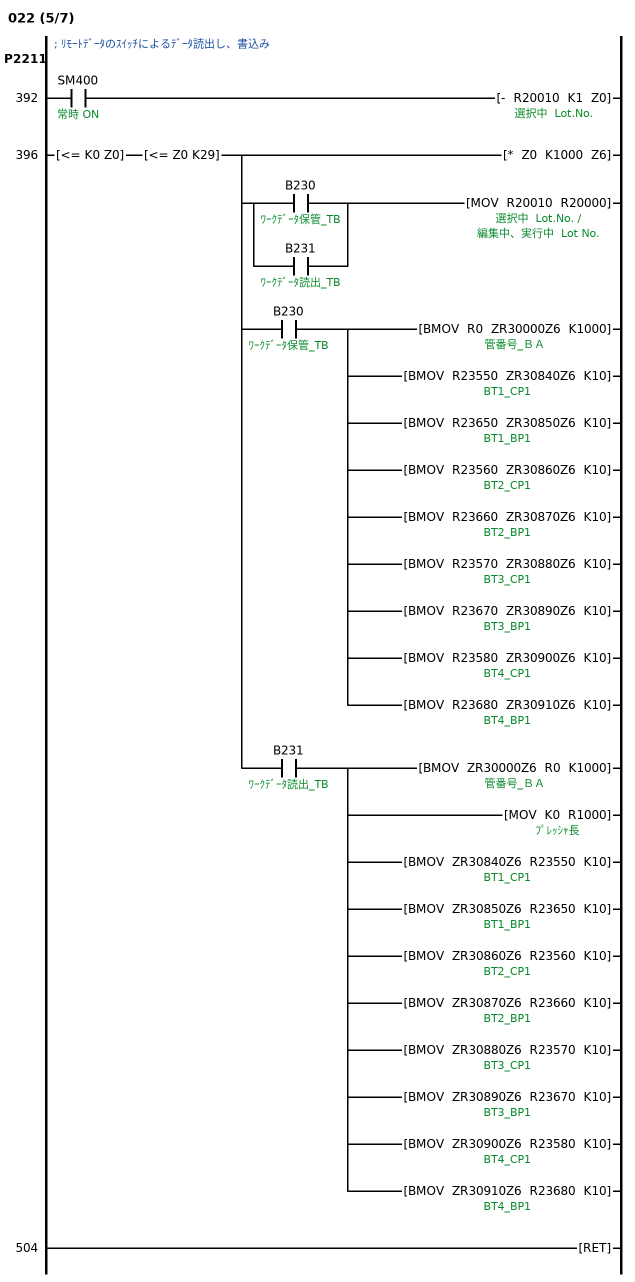
392   LD      SM400  ; 常時 ON
      -       R20010 K1 Z0
396   LD<=    K0 Z0
      AND<=   Z0 K29
      *       Z0 K1000 Z6
      MPS
      LD      B230  ; ﾜｰｸﾃﾞｰﾀ保管_TB
      OR      B231  ; ﾜｰｸﾃﾞｰﾀ読出_TB
      ANB
      MOV     R20010 R20000
      MRD
      AND     B230  ; ﾜｰｸﾃﾞｰﾀ保管_TB
      BMOV    R0 ZR30000Z6 K1000
      BMOV    R23550 ZR30840Z6 K10
      BMOV    R23650 ZR30850Z6 K10
      BMOV    R23560 ZR30860Z6 K10
      BMOV    R23660 ZR30870Z6 K10
      BMOV    R23570 ZR30880Z6 K10
      BMOV    R23670 ZR30890Z6 K10
      BMOV    R23580 ZR30900Z6 K10
      BMOV    R23680 ZR30910Z6 K10
      MPP
      AND     B231  ; ﾜｰｸﾃﾞｰﾀ読出_TB
      BMOV    ZR30000Z6 R0 K1000
      MOV     K0 R1000
      BMOV    ZR30840Z6 R23550 K10
      BMOV    ZR30850Z6 R23650 K10
      BMOV    ZR30860Z6 R23560 K10
      BMOV    ZR30870Z6 R23660 K10
      BMOV    ZR30880Z6 R23570 K10
      BMOV    ZR30890Z6 R23670 K10
      BMOV    ZR30900Z6 R23580 K10
      BMOV    ZR30910Z6 R23680 K10
504   RET
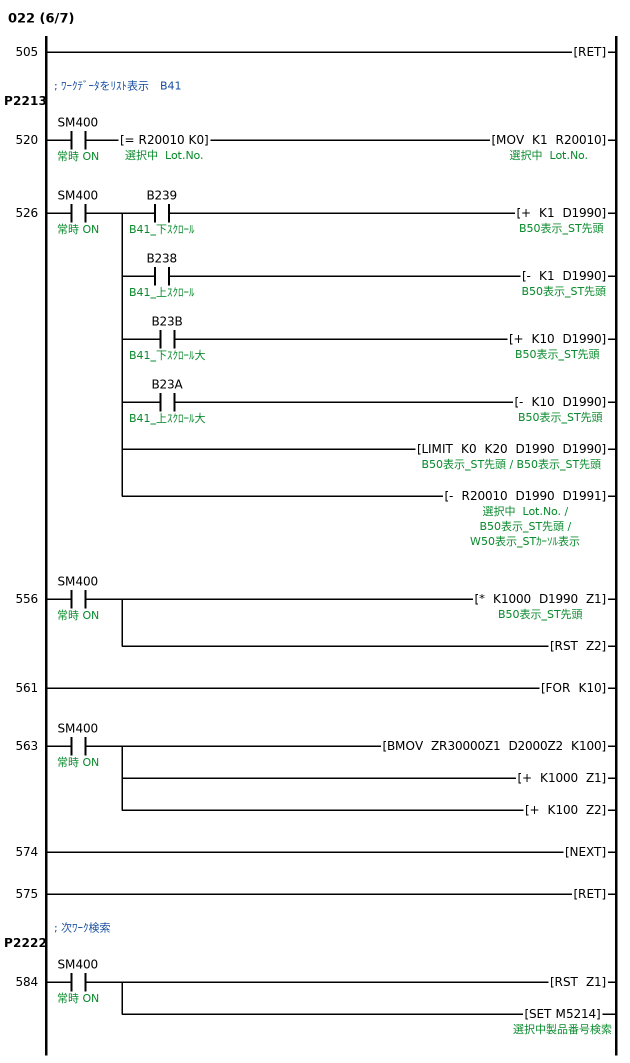
505   RET
; ﾜｰｸﾃﾞｰﾀをﾘｽﾄ表示　B41
      P2213
520   LD      SM400  ; 常時 ON
      AND=    R20010 K0  ; 選択中  Lot.No.
      MOV     K1 R20010
526   LD      SM400  ; 常時 ON
      MPS
      AND     B239  ; B41_下ｽｸﾛｰﾙ
      +       K1 D1990
      MRD
      AND     B238  ; B41_上ｽｸﾛｰﾙ
      -       K1 D1990
      MRD
      AND     B23B  ; B41_下ｽｸﾛｰﾙ大
      +       K10 D1990
      MRD
      AND     B23A  ; B41_上ｽｸﾛｰﾙ大
      -       K10 D1990
      MPP
      LIMIT   K0 K20 D1990 D1990
      -       R20010 D1990 D1991
556   LD      SM400  ; 常時 ON
      *       K1000 D1990 Z1
      RST     Z2
561   FOR     K10
563   LD      SM400  ; 常時 ON
      BMOV    ZR30000Z1 D2000Z2 K100
      +       K1000 Z1
      +       K100 Z2
574   NEXT
575   RET
; 次ﾜｰｸ検索
      P2222
584   LD      SM400  ; 常時 ON
      RST     Z1
      SET     M5214  ; 選択中製品番号検索
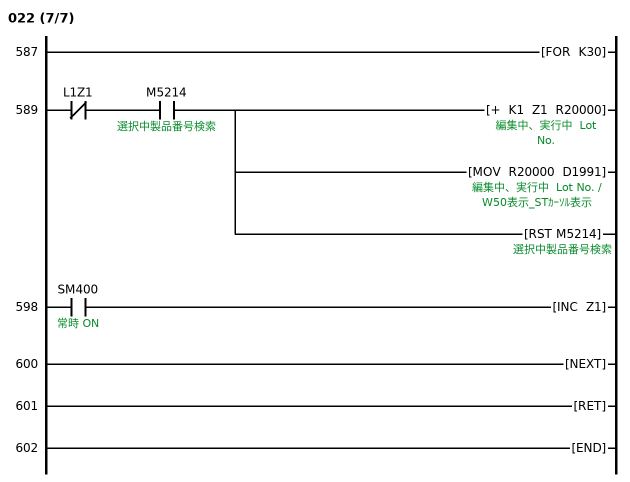
587   FOR     K30
589   LDI     L1Z1
      AND     M5214  ; 選択中製品番号検索
      +       K1 Z1 R20000
      MOV     R20000 D1991
      RST     M5214  ; 選択中製品番号検索
598   LD      SM400  ; 常時 ON
      INC     Z1
600   NEXT
601   RET
602   END
END_PROGRAM

PROGRAM 023  // ﾃﾞｰﾀﾁｪｯｸ
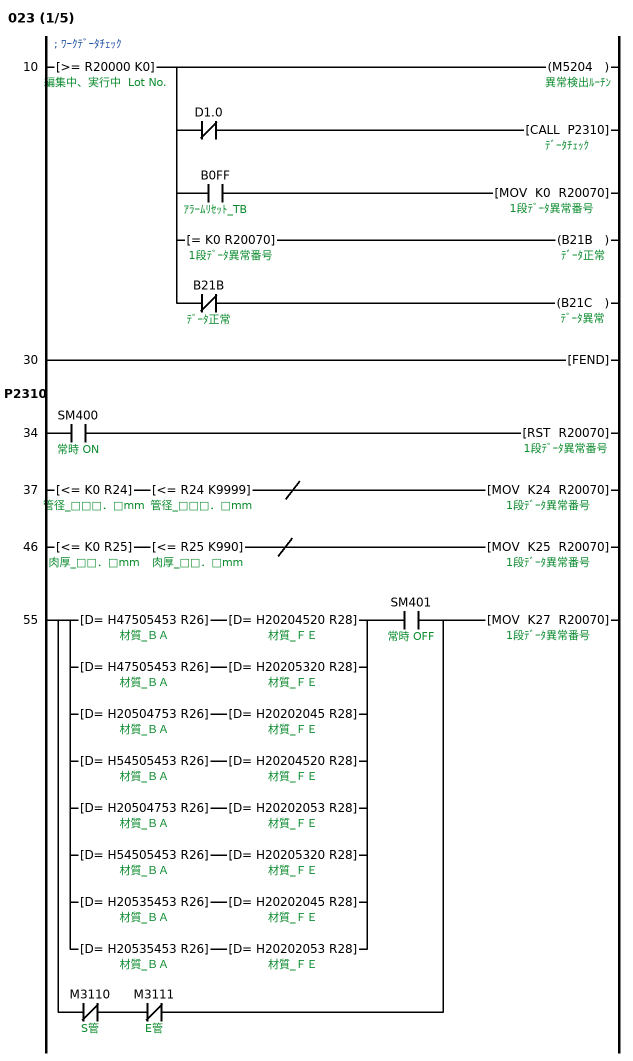
; 
; ﾜｰｸﾃﾞｰﾀﾁｪｯｸ
10    LD>=    R20000 K0  ; 編集中、実行中  Lot No.
      OUT     M5204  ; 異常検出ﾙｰﾁﾝ
      MPS
      ANI     D1.0
      CALL    P2310  ; ﾃﾞｰﾀﾁｪｯｸ
      MRD
      AND     B0FF  ; ｱﾗｰﾑﾘｾｯﾄ_TB
      MOV     K0 R20070  ; 1段ﾃﾞｰﾀ異常番号
      MRD
      AND=    K0 R20070  ; 1段ﾃﾞｰﾀ異常番号
      OUT     B21B  ; ﾃﾞｰﾀ正常
      MPP
      ANI     B21B  ; ﾃﾞｰﾀ正常
      OUT     B21C  ; ﾃﾞｰﾀ異常
30    FEND
; 
      P2310
34    LD      SM400  ; 常時 ON
      RST     R20070  ; 1段ﾃﾞｰﾀ異常番号
37    LD<=    K0 R24  ; 管径_□□□．□mm
      AND<=   R24 K9999  ; 管径_□□□．□mm
      INV
      MOV     K24 R20070
46    LD<=    K0 R25  ; 肉厚_□□．□mm
      AND<=   R25 K990  ; 肉厚_□□．□mm
      INV
      MOV     K25 R20070
55    LDD=    H47505453 R26  ; 材質_ＢＡ
      ANDD=   H20204520 R28  ; 材質_ＦＥ
      LDD=    H47505453 R26  ; 材質_ＢＡ
      ANDD=   H20205320 R28  ; 材質_ＦＥ
      ORB
      LDD=    H20504753 R26  ; 材質_ＢＡ
      ANDD=   H20202045 R28  ; 材質_ＦＥ
      ORB
      LDD=    H54505453 R26  ; 材質_ＢＡ
      ANDD=   H20204520 R28  ; 材質_ＦＥ
      ORB
      LDD=    H20504753 R26  ; 材質_ＢＡ
      ANDD=   H20202053 R28  ; 材質_ＦＥ
      ORB
      LDD=    H54505453 R26  ; 材質_ＢＡ
      ANDD=   H20205320 R28  ; 材質_ＦＥ
      ORB
      LDD=    H20535453 R26  ; 材質_ＢＡ
      ANDD=   H20202045 R28  ; 材質_ＦＥ
      ORB
      LDD=    H20535453 R26  ; 材質_ＢＡ
      ANDD=   H20202053 R28  ; 材質_ＦＥ
      ORB
      AND     SM401  ; 常時 OFF
      LDI     M3110  ; S管
      ANI     M3111  ; E管
      ORB
      MOV     K27 R20070
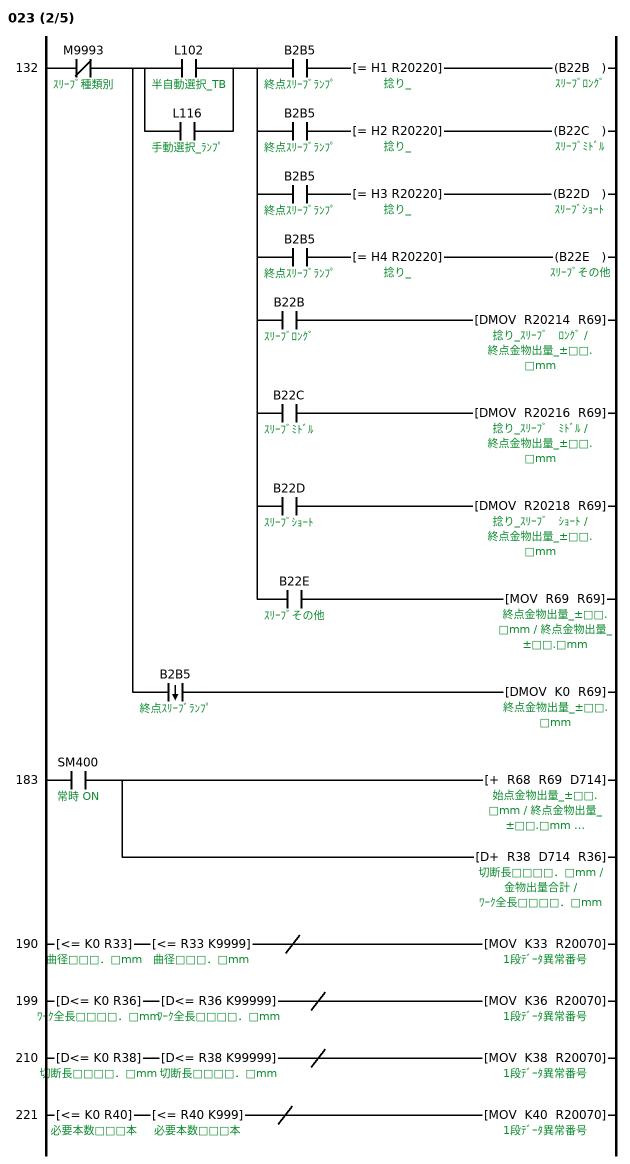
132   LDI     M9993  ; ｽﾘｰﾌﾞ種類別
      MPS
      LD      L102  ; 半自動選択_TB
      OR      L116  ; 手動選択_ﾗﾝﾌﾟ
      ANB
      MPS
      AND     B2B5  ; 終点ｽﾘｰﾌﾞﾗﾝﾌﾟ
      AND=    H1 R20220  ; 捻り_
      OUT     B22B  ; ｽﾘｰﾌﾞﾛﾝｸﾞ
      MRD
      AND     B2B5  ; 終点ｽﾘｰﾌﾞﾗﾝﾌﾟ
      AND=    H2 R20220  ; 捻り_
      OUT     B22C  ; ｽﾘｰﾌﾞﾐﾄﾞﾙ
      MRD
      AND     B2B5  ; 終点ｽﾘｰﾌﾞﾗﾝﾌﾟ
      AND=    H3 R20220  ; 捻り_
      OUT     B22D  ; ｽﾘｰﾌﾞｼｮｰﾄ
      MRD
      AND     B2B5  ; 終点ｽﾘｰﾌﾞﾗﾝﾌﾟ
      AND=    H4 R20220  ; 捻り_
      OUT     B22E  ; ｽﾘｰﾌﾞその他
      MRD
      AND     B22B  ; ｽﾘｰﾌﾞﾛﾝｸﾞ
      DMOV    R20214 R69  ; 捻り_ｽﾘｰﾌﾞ　ﾛﾝｸﾞ / 終点金物出量_±□□.□mm
      MRD
      AND     B22C  ; ｽﾘｰﾌﾞﾐﾄﾞﾙ
      DMOV    R20216 R69  ; 捻り_ｽﾘｰﾌﾞ　ﾐﾄﾞﾙ
      MRD
      AND     B22D  ; ｽﾘｰﾌﾞｼｮｰﾄ
      DMOV    R20218 R69  ; 捻り_ｽﾘｰﾌﾞ　ｼｮｰﾄ
      MPP
      AND     B22E  ; ｽﾘｰﾌﾞその他
      MOV     R69 R69
      MPP
      ANDF    B2B5  ; 終点ｽﾘｰﾌﾞﾗﾝﾌﾟ
      DMOV    K0 R69
183   LD      SM400  ; 常時 ON
      +       R68 R69 D714  ; 始点金物出量_±□□.□mm / 金物出量合計
      D+      R38 D714 R36  ; 切断長□□□□．□mm / ﾜｰｸ全長□□□□．□mm
190   LD<=    K0 R33  ; 曲径□□□．□mm
      AND<=   R33 K9999  ; 曲径□□□．□mm
      INV
      MOV     K33 R20070
199   LDD<=   K0 R36  ; ﾜｰｸ全長□□□□．□mm
      ANDD<=  R36 K99999  ; ﾜｰｸ全長□□□□．□mm
      INV
      MOV     K36 R20070
210   LDD<=   K0 R38  ; 切断長□□□□．□mm
      ANDD<=  R38 K99999  ; 切断長□□□□．□mm
      INV
      MOV     K38 R20070
221   LD<=    K0 R40  ; 必要本数□□□本
      AND<=   R40 K999  ; 必要本数□□□本
      INV
      MOV     K40 R20070
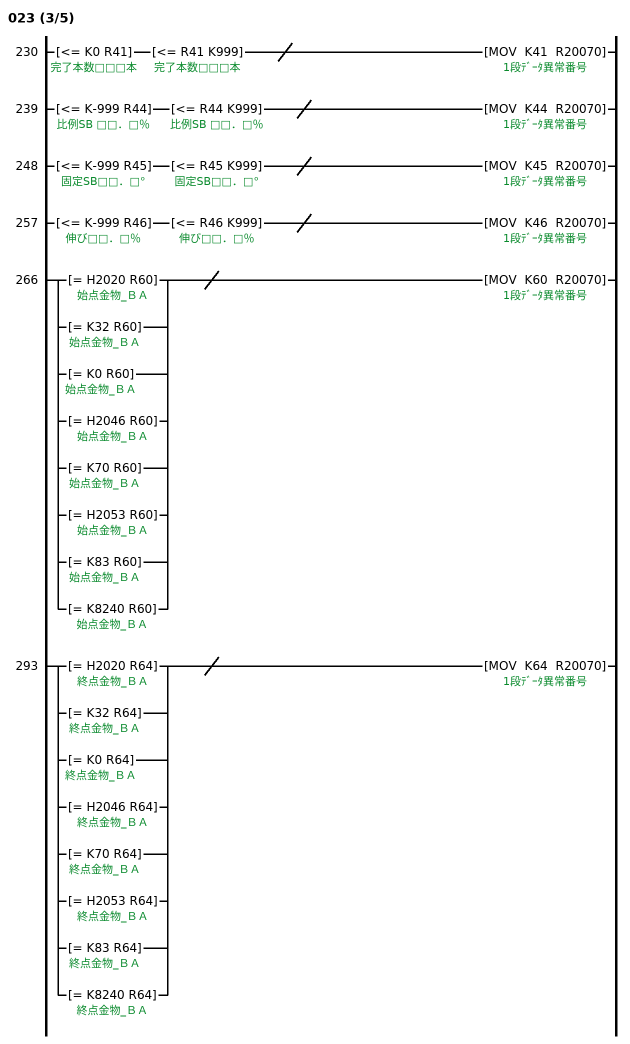
230   LD<=    K0 R41  ; 完了本数□□□本
      AND<=   R41 K999  ; 完了本数□□□本
      INV
      MOV     K41 R20070
239   LD<=    K-999 R44  ; 比例SB □□．□％
      AND<=   R44 K999  ; 比例SB □□．□％
      INV
      MOV     K44 R20070
248   LD<=    K-999 R45  ; 固定SB□□．□°
      AND<=   R45 K999  ; 固定SB□□．□°
      INV
      MOV     K45 R20070
257   LD<=    K-999 R46  ; 伸び□□．□％
      AND<=   R46 K999  ; 伸び□□．□％
      INV
      MOV     K46 R20070
266   LD=     H2020 R60  ; 始点金物_ＢＡ
      OR=     K32 R60  ; 始点金物_ＢＡ
      OR=     K0 R60  ; 始点金物_ＢＡ
      OR=     H2046 R60  ; 始点金物_ＢＡ
      OR=     K70 R60  ; 始点金物_ＢＡ
      OR=     H2053 R60  ; 始点金物_ＢＡ
      OR=     K83 R60  ; 始点金物_ＢＡ
      OR=     K8240 R60  ; 始点金物_ＢＡ
      INV
      MOV     K60 R20070
293   LD=     H2020 R64  ; 終点金物_ＢＡ
      OR=     K32 R64  ; 終点金物_ＢＡ
      OR=     K0 R64  ; 終点金物_ＢＡ
      OR=     H2046 R64  ; 終点金物_ＢＡ
      OR=     K70 R64  ; 終点金物_ＢＡ
      OR=     H2053 R64  ; 終点金物_ＢＡ
      OR=     K83 R64  ; 終点金物_ＢＡ
      OR=     K8240 R64  ; 終点金物_ＢＡ
      INV
      MOV     K64 R20070
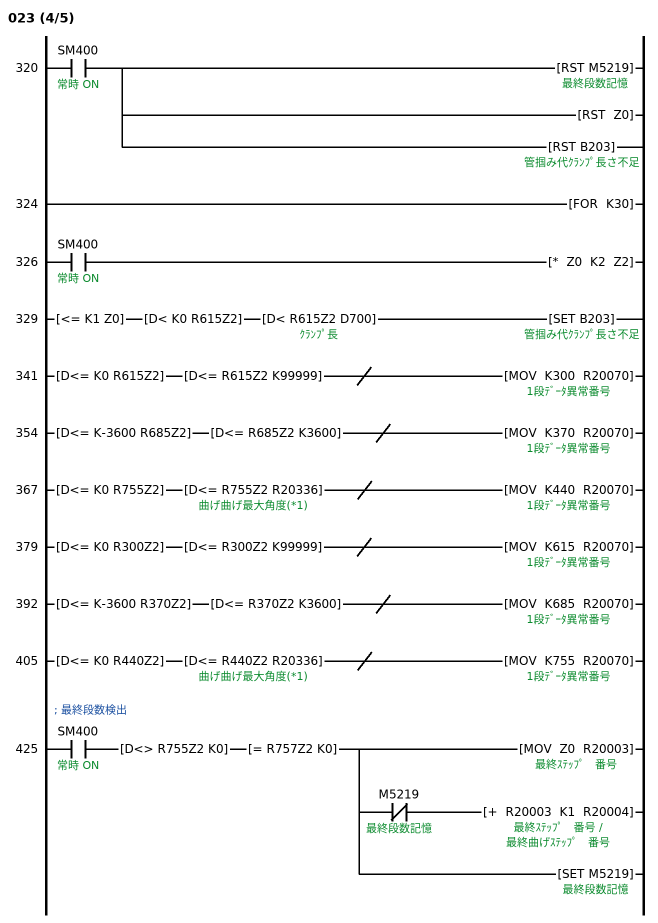
320   LD      SM400  ; 常時 ON
      RST     M5219  ; 最終段数記憶
      RST     Z0
      RST     B203  ; 管掴み代ｸﾗﾝﾌﾟ長さ不足
324   FOR     K30
326   LD      SM400  ; 常時 ON
      *       Z0 K2 Z2
329   LD<=    K1 Z0
      ANDD<   K0 R615Z2
      ANDD<   R615Z2 D700  ; ｸﾗﾝﾌﾟ長
      SET     B203  ; 管掴み代ｸﾗﾝﾌﾟ長さ不足
341   LDD<=   K0 R615Z2
      ANDD<=  R615Z2 K99999
      INV
      MOV     K300 R20070
354   LDD<=   K-3600 R685Z2
      ANDD<=  R685Z2 K3600
      INV
      MOV     K370 R20070
367   LDD<=   K0 R755Z2
      ANDD<=  R755Z2 R20336  ; 曲げ曲げ最大角度(*1)
      INV
      MOV     K440 R20070
379   LDD<=   K0 R300Z2
      ANDD<=  R300Z2 K99999
      INV
      MOV     K615 R20070
392   LDD<=   K-3600 R370Z2
      ANDD<=  R370Z2 K3600
      INV
      MOV     K685 R20070
405   LDD<=   K0 R440Z2
      ANDD<=  R440Z2 R20336  ; 曲げ曲げ最大角度(*1)
      INV
      MOV     K755 R20070
; 最終段数検出
425   LD      SM400  ; 常時 ON
      ANDD<>  R755Z2 K0
      AND=    R757Z2 K0
      MOV     Z0 R20003  ; 最終ｽﾃｯﾌﾟ   番号
      MPS
      ANI     M5219  ; 最終段数記憶
      +       R20003 K1 R20004  ; 最終曲げｽﾃｯﾌﾟ   番号
      MPP
      SET     M5219  ; 最終段数記憶
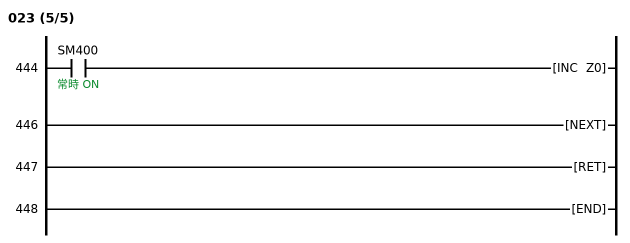
444   LD      SM400  ; 常時 ON
      INC     Z0
446   NEXT
447   RET
448   END
END_PROGRAM

PROGRAM 025  // 完了表示とPC通信
; 完了表示＊Ｙ付加
      P2500
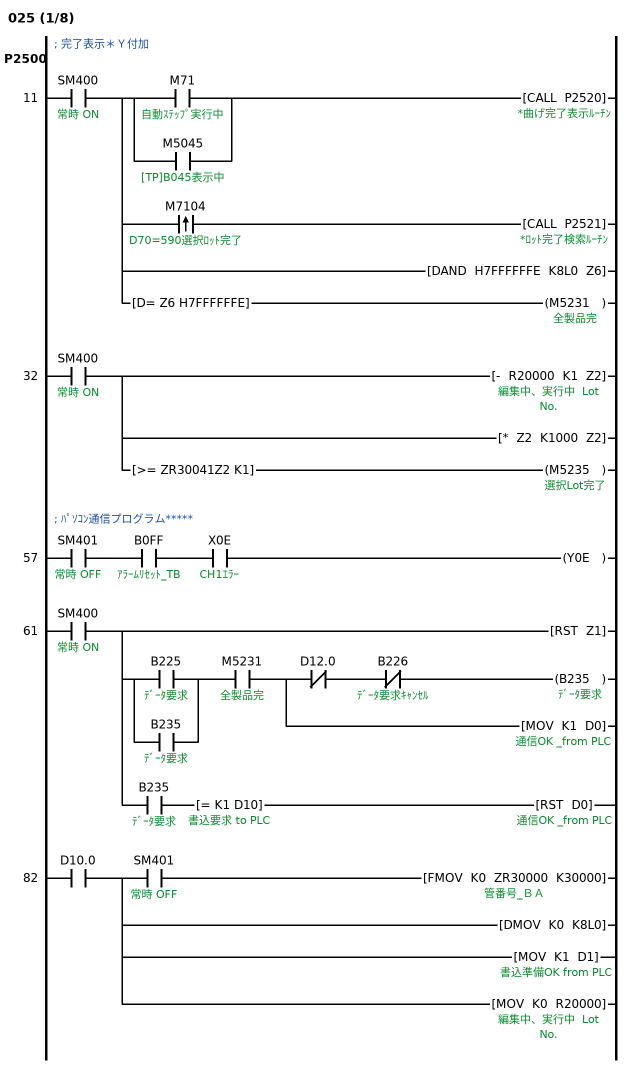
11    LD      SM400  ; 常時 ON
      MPS
      LD      M71  ; 自動ｽﾃｯﾌﾟ実行中
      OR      M5045  ; [TP]B045表示中
      ANB
      CALL    P2520  ; *曲げ完了表示ﾙｰﾁﾝ
      MRD
      ANDP    M7104  ; D70=590選択ﾛｯﾄ完了
      CALL    P2521  ; *ﾛｯﾄ完了検索ﾙｰﾁﾝ
      MPP
      DAND    H7FFFFFFE K8L0 Z6
      ANDD=   Z6 H7FFFFFFE
      OUT     M5231  ; 全製品完
32    LD      SM400  ; 常時 ON
      -       R20000 K1 Z2  ; 編集中、実行中  Lot No.
      *       Z2 K1000 Z2
      AND>=   ZR30041Z2 K1
      OUT     M5235  ; 選択Lot完了
; ﾊﾟｿｺﾝ通信プログラム*****
57    LD      SM401  ; 常時 OFF
      AND     B0FF  ; ｱﾗｰﾑﾘｾｯﾄ_TB
      AND     X0E  ; CH1ｴﾗｰ
      OUT     Y0E
61    LD      SM400  ; 常時 ON
      RST     Z1
      MPS
      LD      B225  ; ﾃﾞｰﾀ要求
      OR      B235  ; ﾃﾞｰﾀ要求
      ANB
      AND     M5231  ; 全製品完
      MPS
      ANI     D12.0
      ANI     B226  ; ﾃﾞｰﾀ要求ｷｬﾝｾﾙ
      OUT     B235  ; ﾃﾞｰﾀ要求
      MPP
      MOV     K1 D0  ; 通信OK _from PLC
      MPP
      AND     B235  ; ﾃﾞｰﾀ要求
      AND=    K1 D10  ; 書込要求 to PLC
      RST     D0  ; 通信OK _from PLC
82    LD      D10.0
      MPS
      AND     SM401  ; 常時 OFF
      FMOV    K0 ZR30000 K30000  ; 管番号_ＢＡ
      MPP
      DMOV    K0 K8L0
      MOV     K1 D1  ; 書込準備OK from PLC
      MOV     K0 R20000
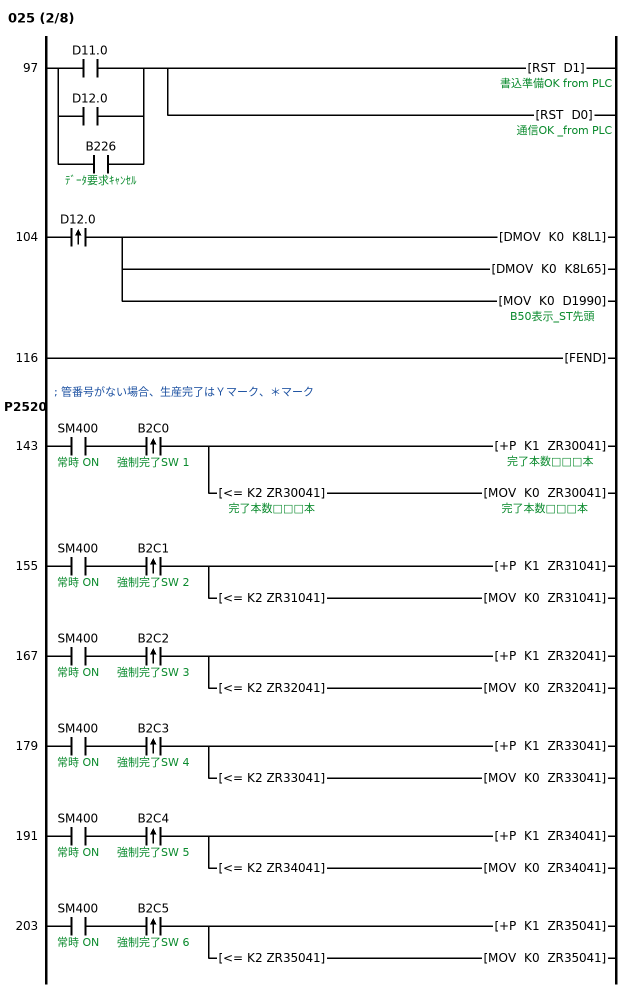
97    LD      D11.0
      OR      D12.0
      OR      B226  ; ﾃﾞｰﾀ要求ｷｬﾝｾﾙ
      RST     D1  ; 書込準備OK from PLC
      RST     D0  ; 通信OK _from PLC
104   LDP     D12.0
      DMOV    K0 K8L1  ; ﾛｯﾄ№-01作業完了
      DMOV    K0 K8L65  ; ﾛｯﾄ№-01作業完了記憶
      MOV     K0 D1990  ; B50表示_ST先頭
116   FEND
; 管番号がない場合、生産完了はＹマーク、＊マーク
      P2520
143   LD      SM400  ; 常時 ON
      ANDP    B2C0  ; 強制完了SW 1
      +P      K1 ZR30041  ; 完了本数□□□本
      AND<=   K2 ZR30041  ; 完了本数□□□本
      MOV     K0 ZR30041
155   LD      SM400  ; 常時 ON
      ANDP    B2C1  ; 強制完了SW 2
      +P      K1 ZR31041
      AND<=   K2 ZR31041
      MOV     K0 ZR31041
167   LD      SM400  ; 常時 ON
      ANDP    B2C2  ; 強制完了SW 3
      +P      K1 ZR32041
      AND<=   K2 ZR32041
      MOV     K0 ZR32041
179   LD      SM400  ; 常時 ON
      ANDP    B2C3  ; 強制完了SW 4
      +P      K1 ZR33041
      AND<=   K2 ZR33041
      MOV     K0 ZR33041
191   LD      SM400  ; 常時 ON
      ANDP    B2C4  ; 強制完了SW 5
      +P      K1 ZR34041
      AND<=   K2 ZR34041
      MOV     K0 ZR34041
203   LD      SM400  ; 常時 ON
      ANDP    B2C5  ; 強制完了SW 6
      +P      K1 ZR35041
      AND<=   K2 ZR35041
      MOV     K0 ZR35041
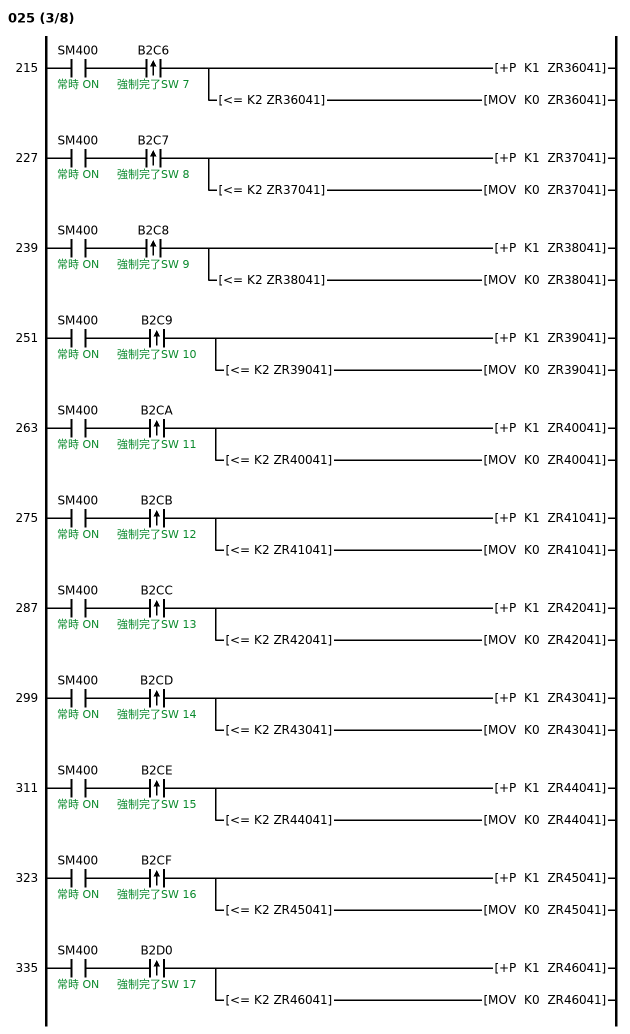
215   LD      SM400  ; 常時 ON
      ANDP    B2C6  ; 強制完了SW 7
      +P      K1 ZR36041
      AND<=   K2 ZR36041
      MOV     K0 ZR36041
227   LD      SM400  ; 常時 ON
      ANDP    B2C7  ; 強制完了SW 8
      +P      K1 ZR37041
      AND<=   K2 ZR37041
      MOV     K0 ZR37041
239   LD      SM400  ; 常時 ON
      ANDP    B2C8  ; 強制完了SW 9
      +P      K1 ZR38041
      AND<=   K2 ZR38041
      MOV     K0 ZR38041
251   LD      SM400  ; 常時 ON
      ANDP    B2C9  ; 強制完了SW 10
      +P      K1 ZR39041
      AND<=   K2 ZR39041
      MOV     K0 ZR39041
263   LD      SM400  ; 常時 ON
      ANDP    B2CA  ; 強制完了SW 11
      +P      K1 ZR40041
      AND<=   K2 ZR40041
      MOV     K0 ZR40041
275   LD      SM400  ; 常時 ON
      ANDP    B2CB  ; 強制完了SW 12
      +P      K1 ZR41041
      AND<=   K2 ZR41041
      MOV     K0 ZR41041
287   LD      SM400  ; 常時 ON
      ANDP    B2CC  ; 強制完了SW 13
      +P      K1 ZR42041
      AND<=   K2 ZR42041
      MOV     K0 ZR42041
299   LD      SM400  ; 常時 ON
      ANDP    B2CD  ; 強制完了SW 14
      +P      K1 ZR43041
      AND<=   K2 ZR43041
      MOV     K0 ZR43041
311   LD      SM400  ; 常時 ON
      ANDP    B2CE  ; 強制完了SW 15
      +P      K1 ZR44041
      AND<=   K2 ZR44041
      MOV     K0 ZR44041
323   LD      SM400  ; 常時 ON
      ANDP    B2CF  ; 強制完了SW 16
      +P      K1 ZR45041
      AND<=   K2 ZR45041
      MOV     K0 ZR45041
335   LD      SM400  ; 常時 ON
      ANDP    B2D0  ; 強制完了SW 17
      +P      K1 ZR46041
      AND<=   K2 ZR46041
      MOV     K0 ZR46041
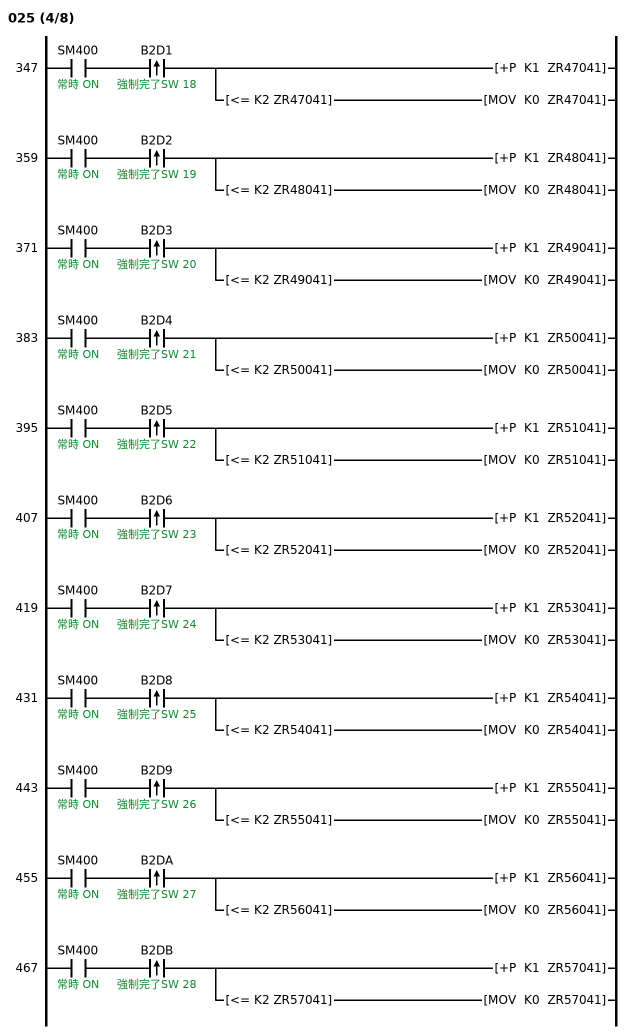
347   LD      SM400  ; 常時 ON
      ANDP    B2D1  ; 強制完了SW 18
      +P      K1 ZR47041
      AND<=   K2 ZR47041
      MOV     K0 ZR47041
359   LD      SM400  ; 常時 ON
      ANDP    B2D2  ; 強制完了SW 19
      +P      K1 ZR48041
      AND<=   K2 ZR48041
      MOV     K0 ZR48041
371   LD      SM400  ; 常時 ON
      ANDP    B2D3  ; 強制完了SW 20
      +P      K1 ZR49041
      AND<=   K2 ZR49041
      MOV     K0 ZR49041
383   LD      SM400  ; 常時 ON
      ANDP    B2D4  ; 強制完了SW 21
      +P      K1 ZR50041
      AND<=   K2 ZR50041
      MOV     K0 ZR50041
395   LD      SM400  ; 常時 ON
      ANDP    B2D5  ; 強制完了SW 22
      +P      K1 ZR51041
      AND<=   K2 ZR51041
      MOV     K0 ZR51041
407   LD      SM400  ; 常時 ON
      ANDP    B2D6  ; 強制完了SW 23
      +P      K1 ZR52041
      AND<=   K2 ZR52041
      MOV     K0 ZR52041
419   LD      SM400  ; 常時 ON
      ANDP    B2D7  ; 強制完了SW 24
      +P      K1 ZR53041
      AND<=   K2 ZR53041
      MOV     K0 ZR53041
431   LD      SM400  ; 常時 ON
      ANDP    B2D8  ; 強制完了SW 25
      +P      K1 ZR54041
      AND<=   K2 ZR54041
      MOV     K0 ZR54041
443   LD      SM400  ; 常時 ON
      ANDP    B2D9  ; 強制完了SW 26
      +P      K1 ZR55041
      AND<=   K2 ZR55041
      MOV     K0 ZR55041
455   LD      SM400  ; 常時 ON
      ANDP    B2DA  ; 強制完了SW 27
      +P      K1 ZR56041
      AND<=   K2 ZR56041
      MOV     K0 ZR56041
467   LD      SM400  ; 常時 ON
      ANDP    B2DB  ; 強制完了SW 28
      +P      K1 ZR57041
      AND<=   K2 ZR57041
      MOV     K0 ZR57041
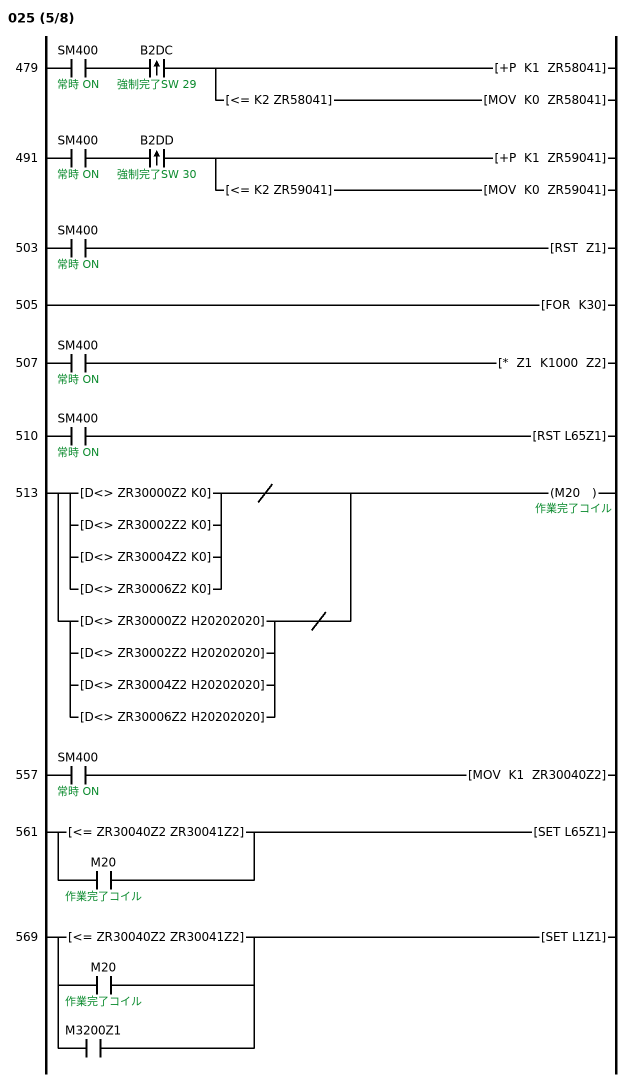
479   LD      SM400  ; 常時 ON
      ANDP    B2DC  ; 強制完了SW 29
      +P      K1 ZR58041
      AND<=   K2 ZR58041
      MOV     K0 ZR58041
491   LD      SM400  ; 常時 ON
      ANDP    B2DD  ; 強制完了SW 30
      +P      K1 ZR59041
      AND<=   K2 ZR59041
      MOV     K0 ZR59041
503   LD      SM400  ; 常時 ON
      RST     Z1
505   FOR     K30
507   LD      SM400  ; 常時 ON
      *       Z1 K1000 Z2
510   LD      SM400  ; 常時 ON
      RST     L65Z1
513   LDD<>   ZR30000Z2 K0
      ORD<>   ZR30002Z2 K0
      ORD<>   ZR30004Z2 K0
      ORD<>   ZR30006Z2 K0
      INV
      LDD<>   ZR30000Z2 H20202020
      ORD<>   ZR30002Z2 H20202020
      ORD<>   ZR30004Z2 H20202020
      ORD<>   ZR30006Z2 H20202020
      INV
      ORB
      OUT     M20  ; 作業完了コイル
557   LD      SM400  ; 常時 ON
      MOV     K1 ZR30040Z2
561   LD<=    ZR30040Z2 ZR30041Z2
      OR      M20  ; 作業完了コイル
      SET     L65Z1
569   LD<=    ZR30040Z2 ZR30041Z2
      OR      M20  ; 作業完了コイル
      OR      M3200Z1
      SET     L1Z1
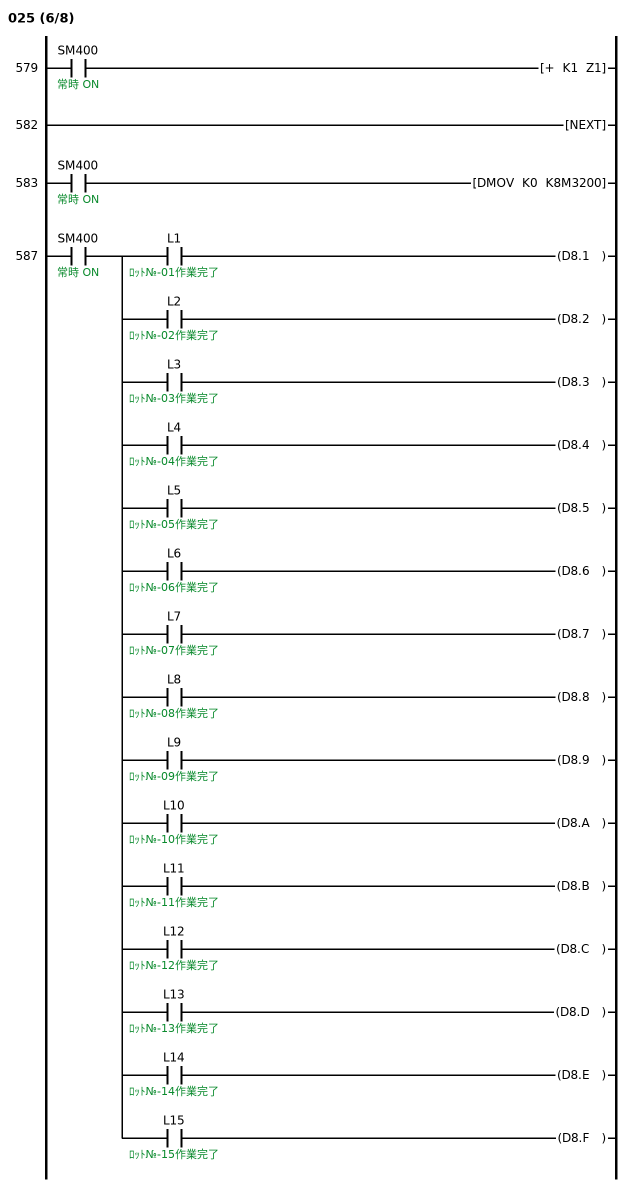
579   LD      SM400  ; 常時 ON
      +       K1 Z1
582   NEXT
583   LD      SM400  ; 常時 ON
      DMOV    K0 K8M3200  ; ﾛｯﾄNo.-01作業完了
587   LD      SM400  ; 常時 ON
      MPS
      AND     L1  ; ﾛｯﾄ№-01作業完了
      OUT     D8.1
      MRD
      AND     L2  ; ﾛｯﾄ№-02作業完了
      OUT     D8.2
      MRD
      AND     L3  ; ﾛｯﾄ№-03作業完了
      OUT     D8.3
      MRD
      AND     L4  ; ﾛｯﾄ№-04作業完了
      OUT     D8.4
      MRD
      AND     L5  ; ﾛｯﾄ№-05作業完了
      OUT     D8.5
      MRD
      AND     L6  ; ﾛｯﾄ№-06作業完了
      OUT     D8.6
      MRD
      AND     L7  ; ﾛｯﾄ№-07作業完了
      OUT     D8.7
      MRD
      AND     L8  ; ﾛｯﾄ№-08作業完了
      OUT     D8.8
      MRD
      AND     L9  ; ﾛｯﾄ№-09作業完了
      OUT     D8.9
      MRD
      AND     L10  ; ﾛｯﾄ№-10作業完了
      OUT     D8.A
      MRD
      AND     L11  ; ﾛｯﾄ№-11作業完了
      OUT     D8.B
      MRD
      AND     L12  ; ﾛｯﾄ№-12作業完了
      OUT     D8.C
      MRD
      AND     L13  ; ﾛｯﾄ№-13作業完了
      OUT     D8.D
      MRD
      AND     L14  ; ﾛｯﾄ№-14作業完了
      OUT     D8.E
      MPP
      AND     L15  ; ﾛｯﾄ№-15作業完了
      OUT     D8.F
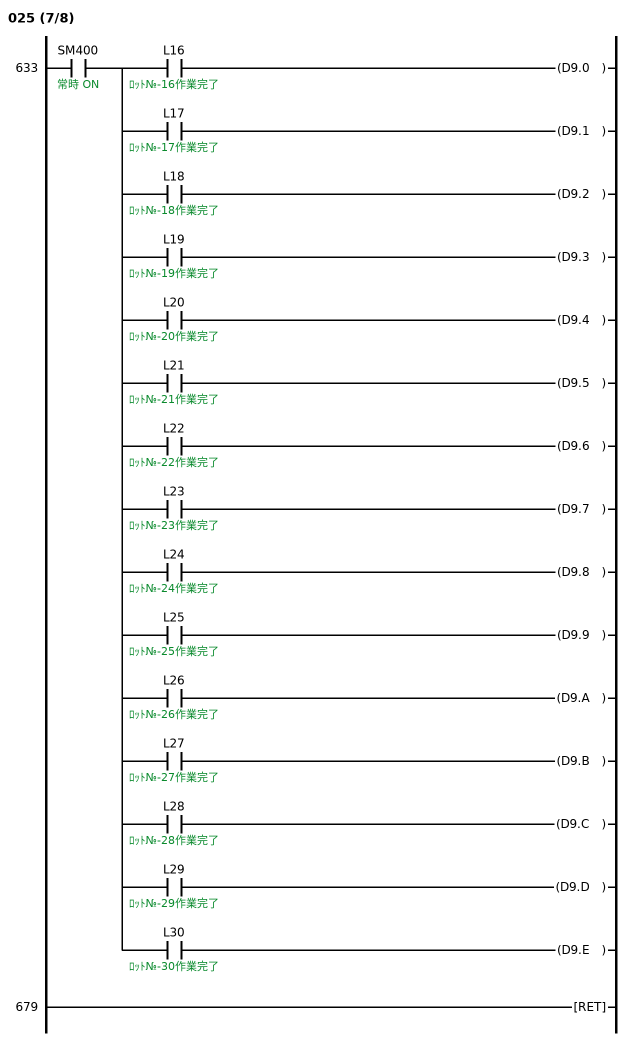
633   LD      SM400  ; 常時 ON
      MPS
      AND     L16  ; ﾛｯﾄ№-16作業完了
      OUT     D9.0
      MRD
      AND     L17  ; ﾛｯﾄ№-17作業完了
      OUT     D9.1
      MRD
      AND     L18  ; ﾛｯﾄ№-18作業完了
      OUT     D9.2
      MRD
      AND     L19  ; ﾛｯﾄ№-19作業完了
      OUT     D9.3
      MRD
      AND     L20  ; ﾛｯﾄ№-20作業完了
      OUT     D9.4
      MRD
      AND     L21  ; ﾛｯﾄ№-21作業完了
      OUT     D9.5
      MRD
      AND     L22  ; ﾛｯﾄ№-22作業完了
      OUT     D9.6
      MRD
      AND     L23  ; ﾛｯﾄ№-23作業完了
      OUT     D9.7
      MRD
      AND     L24  ; ﾛｯﾄ№-24作業完了
      OUT     D9.8
      MRD
      AND     L25  ; ﾛｯﾄ№-25作業完了
      OUT     D9.9
      MRD
      AND     L26  ; ﾛｯﾄ№-26作業完了
      OUT     D9.A
      MRD
      AND     L27  ; ﾛｯﾄ№-27作業完了
      OUT     D9.B
      MRD
      AND     L28  ; ﾛｯﾄ№-28作業完了
      OUT     D9.C
      MRD
      AND     L29  ; ﾛｯﾄ№-29作業完了
      OUT     D9.D
      MPP
      AND     L30  ; ﾛｯﾄ№-30作業完了
      OUT     D9.E
679   RET
; 生産本数分完了で完了マーク
      P2521
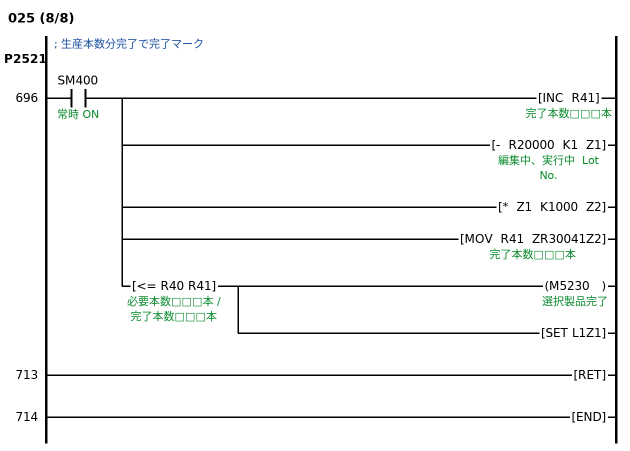
696   LD      SM400  ; 常時 ON
      INC     R41  ; 完了本数□□□本
      -       R20000 K1 Z1
      *       Z1 K1000 Z2
      MOV     R41 ZR30041Z2
      AND<=   R40 R41  ; 必要本数□□□本 / 完了本数□□□本
      OUT     M5230  ; 選択製品完了
      SET     L1Z1
713   RET
714   END
END_PROGRAM

PROGRAM 027  // 管径別ﾃﾞｰﾀ検索
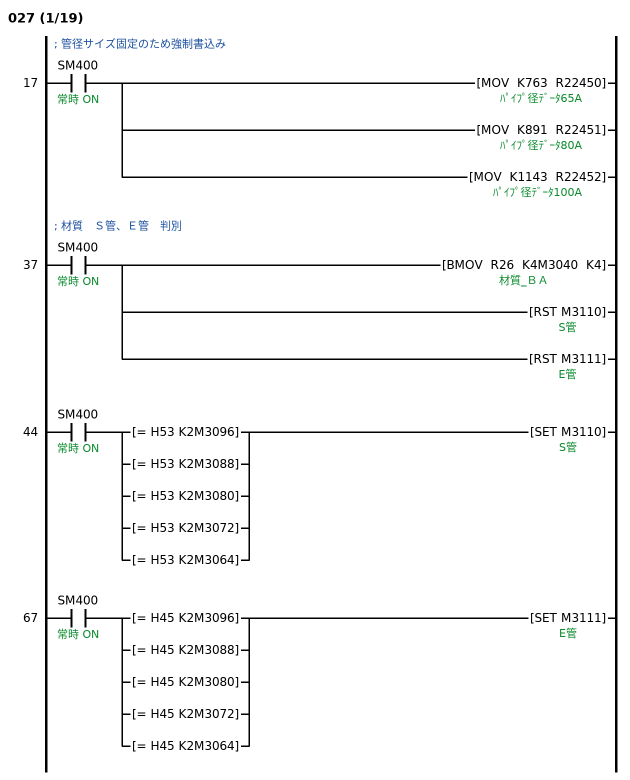
; 管径サイズ固定のため強制書込み
17    LD      SM400  ; 常時 ON
      MOV     K763 R22450  ; ﾊﾟｲﾌﾟ径ﾃﾞｰﾀ65A
      MOV     K891 R22451  ; ﾊﾟｲﾌﾟ径ﾃﾞｰﾀ80A
      MOV     K1143 R22452  ; ﾊﾟｲﾌﾟ径ﾃﾞｰﾀ100A
; 材質　Ｓ管、Ｅ管　判別
37    LD      SM400  ; 常時 ON
      BMOV    R26 K4M3040 K4  ; 材質_ＢＡ / 材質ASCIIﾋﾞｯﾄ置換1
      RST     M3110  ; S管
      RST     M3111  ; E管
44    LD      SM400  ; 常時 ON
      LD=     H53 K2M3096  ; 材質ASCIIﾋﾞｯﾄ置換8
      OR=     H53 K2M3088  ; 材質ASCIIﾋﾞｯﾄ置換7
      OR=     H53 K2M3080  ; 材質ASCIIﾋﾞｯﾄ置換6
      OR=     H53 K2M3072  ; 材質ASCIIﾋﾞｯﾄ置換5
      OR=     H53 K2M3064  ; 材質ASCIIﾋﾞｯﾄ置換4
      ANB
      SET     M3110  ; S管
67    LD      SM400  ; 常時 ON
      LD=     H45 K2M3096  ; 材質ASCIIﾋﾞｯﾄ置換8
      OR=     H45 K2M3088  ; 材質ASCIIﾋﾞｯﾄ置換7
      OR=     H45 K2M3080  ; 材質ASCIIﾋﾞｯﾄ置換6
      OR=     H45 K2M3072  ; 材質ASCIIﾋﾞｯﾄ置換5
      OR=     H45 K2M3064  ; 材質ASCIIﾋﾞｯﾄ置換4
      ANB
      SET     M3111  ; E管
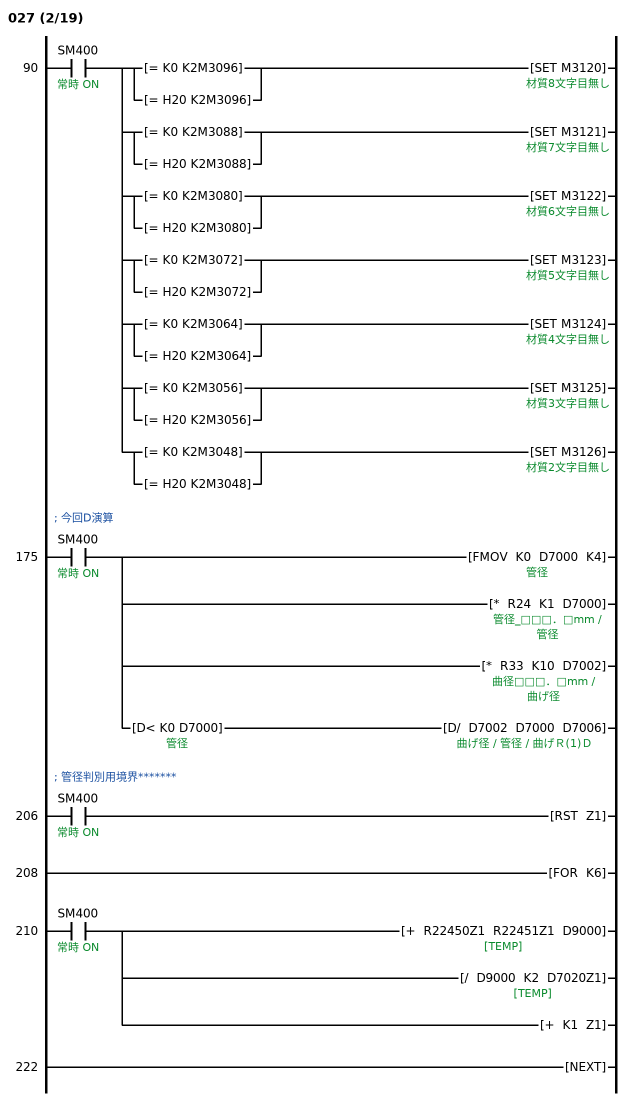
90    LD      SM400  ; 常時 ON
      MPS
      LD=     K0 K2M3096  ; 材質ASCIIﾋﾞｯﾄ置換8
      OR=     H20 K2M3096  ; 材質ASCIIﾋﾞｯﾄ置換8
      ANB
      SET     M3120  ; 材質8文字目無し
      MRD
      LD=     K0 K2M3088  ; 材質ASCIIﾋﾞｯﾄ置換7
      OR=     H20 K2M3088  ; 材質ASCIIﾋﾞｯﾄ置換7
      ANB
      SET     M3121  ; 材質7文字目無し
      MRD
      LD=     K0 K2M3080  ; 材質ASCIIﾋﾞｯﾄ置換6
      OR=     H20 K2M3080  ; 材質ASCIIﾋﾞｯﾄ置換6
      ANB
      SET     M3122  ; 材質6文字目無し
      MRD
      LD=     K0 K2M3072  ; 材質ASCIIﾋﾞｯﾄ置換5
      OR=     H20 K2M3072  ; 材質ASCIIﾋﾞｯﾄ置換5
      ANB
      SET     M3123  ; 材質5文字目無し
      MRD
      LD=     K0 K2M3064  ; 材質ASCIIﾋﾞｯﾄ置換4
      OR=     H20 K2M3064  ; 材質ASCIIﾋﾞｯﾄ置換4
      ANB
      SET     M3124  ; 材質4文字目無し
      MRD
      LD=     K0 K2M3056  ; 材質ASCIIﾋﾞｯﾄ置換3
      OR=     H20 K2M3056  ; 材質ASCIIﾋﾞｯﾄ置換3
      ANB
      SET     M3125  ; 材質3文字目無し
      MPP
      LD=     K0 K2M3048  ; 材質ASCIIﾋﾞｯﾄ置換2
      OR=     H20 K2M3048  ; 材質ASCIIﾋﾞｯﾄ置換2
      ANB
      SET     M3126  ; 材質2文字目無し
; 今回D演算
175   LD      SM400  ; 常時 ON
      FMOV    K0 D7000 K4  ; 管径
      *       R24 K1 D7000  ; 管径_□□□．□mm
      *       R33 K10 D7002  ; 曲径□□□．□mm / 曲げ径
      ANDD<   K0 D7000  ; 管径
      D/      D7002 D7000 D7006  ; 曲げＲ(1)Ｄ
; 管径判別用境界*******
206   LD      SM400  ; 常時 ON
      RST     Z1
208   FOR     K6
210   LD      SM400  ; 常時 ON
      +       R22450Z1 R22451Z1 D9000  ; [TEMP]
      /       D9000 K2 D7020Z1
      +       K1 Z1
222   NEXT
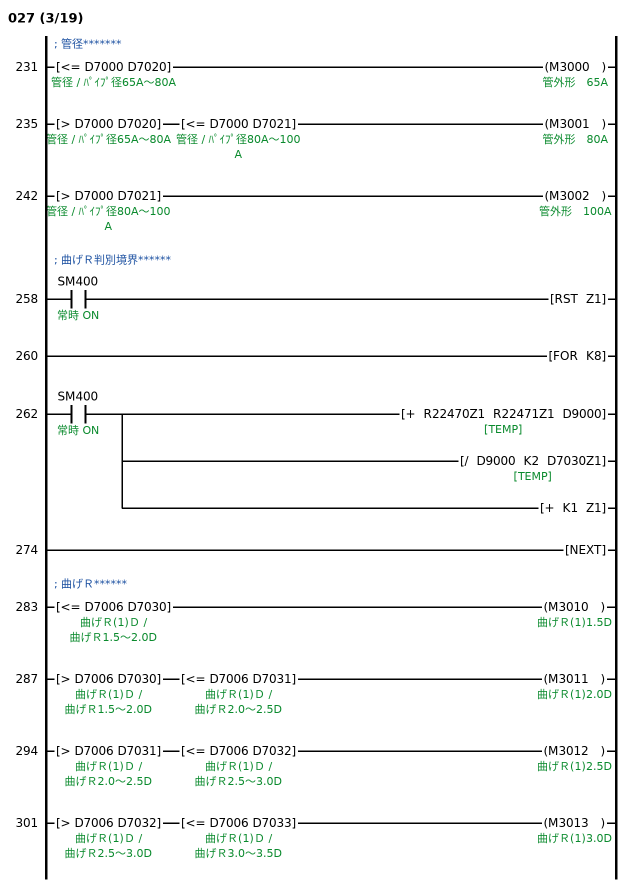
; 管径*******
231   LD<=    D7000 D7020  ; 管径 / ﾊﾟｲﾌﾟ径65A～80A
      OUT     M3000  ; 管外形　65A
235   LD>     D7000 D7020  ; 管径 / ﾊﾟｲﾌﾟ径65A～80A
      AND<=   D7000 D7021  ; 管径 / ﾊﾟｲﾌﾟ径80A～100A
      OUT     M3001  ; 管外形　80A
242   LD>     D7000 D7021  ; 管径 / ﾊﾟｲﾌﾟ径80A～100A
      OUT     M3002  ; 管外形　100A
; 曲げＲ判別境界******
258   LD      SM400  ; 常時 ON
      RST     Z1
260   FOR     K8
262   LD      SM400  ; 常時 ON
      +       R22470Z1 R22471Z1 D9000
      /       D9000 K2 D7030Z1
      +       K1 Z1
274   NEXT
; 曲げＲ******
283   LD<=    D7006 D7030  ; 曲げＲ(1)Ｄ / 曲げＲ1.5～2.0D
      OUT     M3010  ; 曲げＲ(1)1.5D
287   LD>     D7006 D7030  ; 曲げＲ(1)Ｄ / 曲げＲ1.5～2.0D
      AND<=   D7006 D7031  ; 曲げＲ(1)Ｄ / 曲げＲ2.0～2.5D
      OUT     M3011  ; 曲げＲ(1)2.0D
294   LD>     D7006 D7031  ; 曲げＲ(1)Ｄ / 曲げＲ2.0～2.5D
      AND<=   D7006 D7032  ; 曲げＲ(1)Ｄ / 曲げＲ2.5～3.0D
      OUT     M3012  ; 曲げＲ(1)2.5D
301   LD>     D7006 D7032  ; 曲げＲ(1)Ｄ / 曲げＲ2.5～3.0D
      AND<=   D7006 D7033  ; 曲げＲ(1)Ｄ / 曲げＲ3.0～3.5D
      OUT     M3013  ; 曲げＲ(1)3.0D
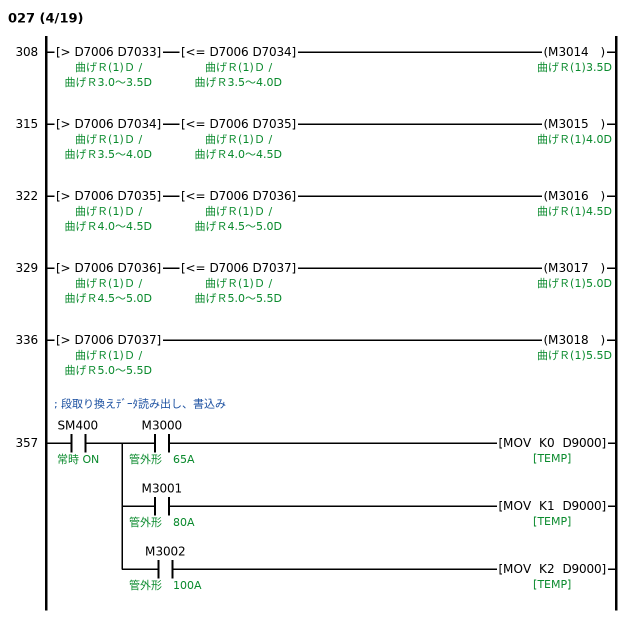
308   LD>     D7006 D7033  ; 曲げＲ(1)Ｄ / 曲げＲ3.0～3.5D
      AND<=   D7006 D7034  ; 曲げＲ(1)Ｄ / 曲げＲ3.5～4.0D
      OUT     M3014  ; 曲げＲ(1)3.5D
315   LD>     D7006 D7034  ; 曲げＲ(1)Ｄ / 曲げＲ3.5～4.0D
      AND<=   D7006 D7035  ; 曲げＲ(1)Ｄ / 曲げＲ4.0～4.5D
      OUT     M3015  ; 曲げＲ(1)4.0D
322   LD>     D7006 D7035  ; 曲げＲ(1)Ｄ / 曲げＲ4.0～4.5D
      AND<=   D7006 D7036  ; 曲げＲ(1)Ｄ / 曲げＲ4.5～5.0D
      OUT     M3016  ; 曲げＲ(1)4.5D
329   LD>     D7006 D7036  ; 曲げＲ(1)Ｄ / 曲げＲ4.5～5.0D
      AND<=   D7006 D7037  ; 曲げＲ(1)Ｄ / 曲げＲ5.0～5.5D
      OUT     M3017  ; 曲げＲ(1)5.0D
336   LD>     D7006 D7037  ; 曲げＲ(1)Ｄ / 曲げＲ5.0～5.5D
      OUT     M3018  ; 曲げＲ(1)5.5D
; 段取り換えﾃﾞｰﾀ読み出し、書込み
357   LD      SM400  ; 常時 ON
      MPS
      AND     M3000  ; 管外形　65A
      MOV     K0 D9000
      MRD
      AND     M3001  ; 管外形　80A
      MOV     K1 D9000
      MPP
      AND     M3002  ; 管外形　100A
      MOV     K2 D9000
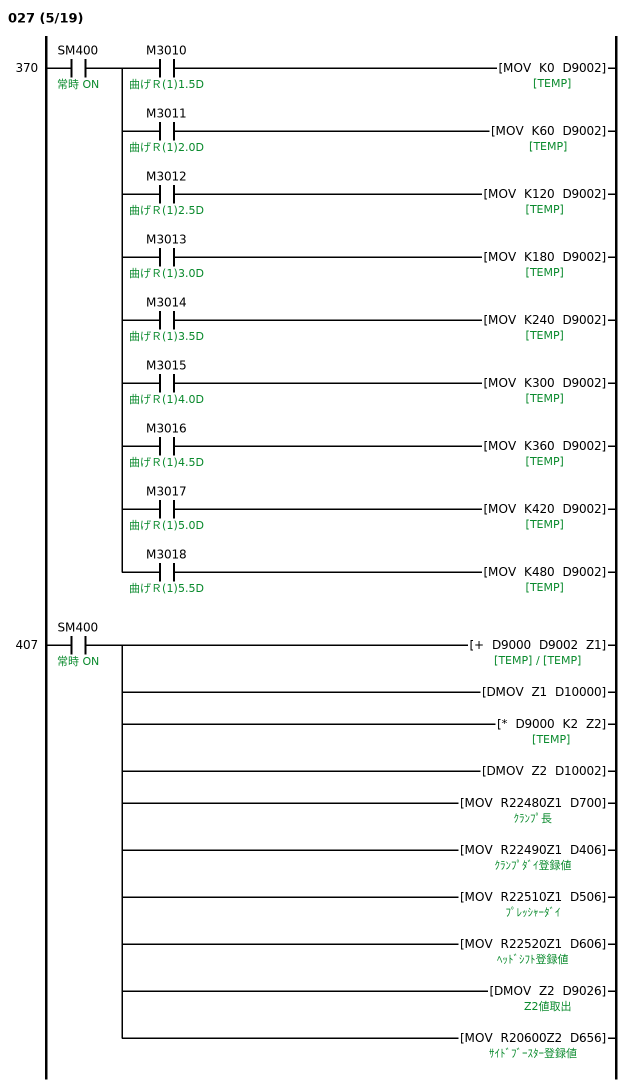
370   LD      SM400  ; 常時 ON
      MPS
      AND     M3010  ; 曲げＲ(1)1.5D
      MOV     K0 D9002  ; [TEMP]
      MRD
      AND     M3011  ; 曲げＲ(1)2.0D
      MOV     K60 D9002
      MRD
      AND     M3012  ; 曲げＲ(1)2.5D
      MOV     K120 D9002
      MRD
      AND     M3013  ; 曲げＲ(1)3.0D
      MOV     K180 D9002
      MRD
      AND     M3014  ; 曲げＲ(1)3.5D
      MOV     K240 D9002
      MRD
      AND     M3015  ; 曲げＲ(1)4.0D
      MOV     K300 D9002
      MRD
      AND     M3016  ; 曲げＲ(1)4.5D
      MOV     K360 D9002
      MRD
      AND     M3017  ; 曲げＲ(1)5.0D
      MOV     K420 D9002
      MPP
      AND     M3018  ; 曲げＲ(1)5.5D
      MOV     K480 D9002
407   LD      SM400  ; 常時 ON
      +       D9000 D9002 Z1
      DMOV    Z1 D10000
      *       D9000 K2 Z2
      DMOV    Z2 D10002
      MOV     R22480Z1 D700  ; ｸﾗﾝﾌﾟ長
      MOV     R22490Z1 D406  ; ｸﾗﾝﾌﾟﾀﾞｲ登録値
      MOV     R22510Z1 D506  ; ﾌﾟﾚｯｼｬｰﾀﾞｲ
      MOV     R22520Z1 D606  ; ﾍｯﾄﾞｼﾌﾄ登録値
      DMOV    Z2 D9026  ; Z2値取出
      MOV     R20600Z2 D656  ; ｻｲﾄﾞﾌﾞｰｽﾀｰ登録値
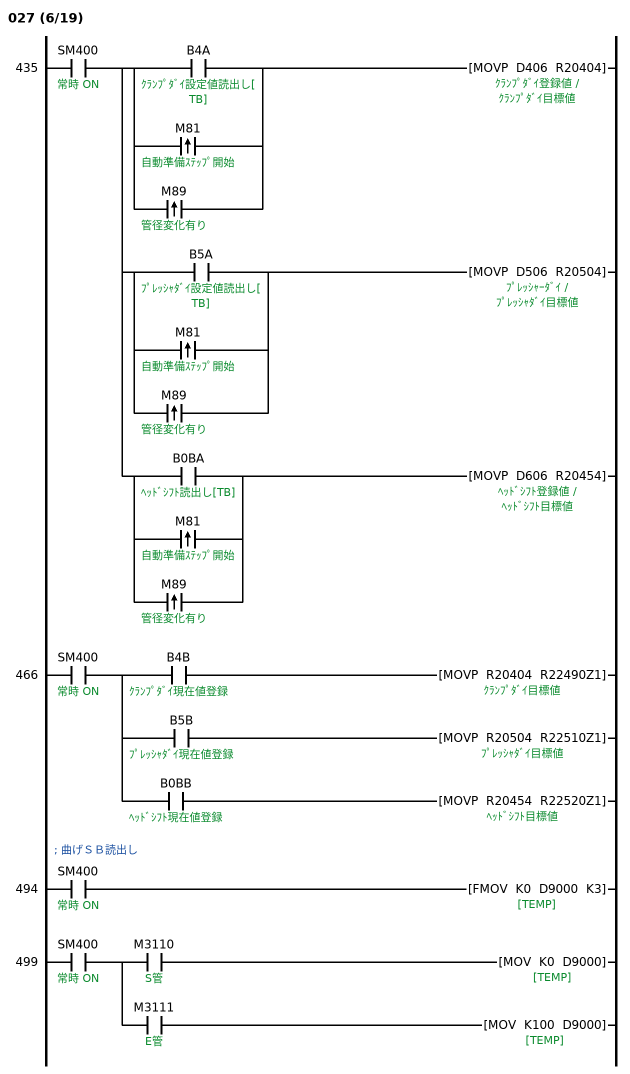
435   LD      SM400  ; 常時 ON
      MPS
      LD      B4A  ; ｸﾗﾝﾌﾟﾀﾞｲ設定値読出し[TB]
      ORP     M81  ; 自動準備ｽﾃｯﾌﾟ開始
      ORP     M89  ; 管径変化有り
      ANB
      MOVP    D406 R20404  ; ｸﾗﾝﾌﾟﾀﾞｲ目標値
      MRD
      LD      B5A  ; ﾌﾟﾚｯｼｬﾀﾞｲ設定値読出し[TB]
      ORP     M81  ; 自動準備ｽﾃｯﾌﾟ開始
      ORP     M89  ; 管径変化有り
      ANB
      MOVP    D506 R20504  ; ﾌﾟﾚｯｼｬﾀﾞｲ目標値
      MPP
      LD      B0BA  ; ﾍｯﾄﾞｼﾌﾄ読出し[TB]
      ORP     M81  ; 自動準備ｽﾃｯﾌﾟ開始
      ORP     M89  ; 管径変化有り
      ANB
      MOVP    D606 R20454  ; ﾍｯﾄﾞｼﾌﾄ目標値
466   LD      SM400  ; 常時 ON
      MPS
      AND     B4B  ; ｸﾗﾝﾌﾟﾀﾞｲ現在値登録
      MOVP    R20404 R22490Z1
      MRD
      AND     B5B  ; ﾌﾟﾚｯｼｬﾀﾞｲ現在値登録
      MOVP    R20504 R22510Z1
      MPP
      AND     B0BB  ; ﾍｯﾄﾞｼﾌﾄ現在値登録
      MOVP    R20454 R22520Z1
; 曲げＳＢ読出し
494   LD      SM400  ; 常時 ON
      FMOV    K0 D9000 K3
499   LD      SM400  ; 常時 ON
      MPS
      AND     M3110  ; S管
      MOV     K0 D9000
      MPP
      AND     M3111  ; E管
      MOV     K100 D9000
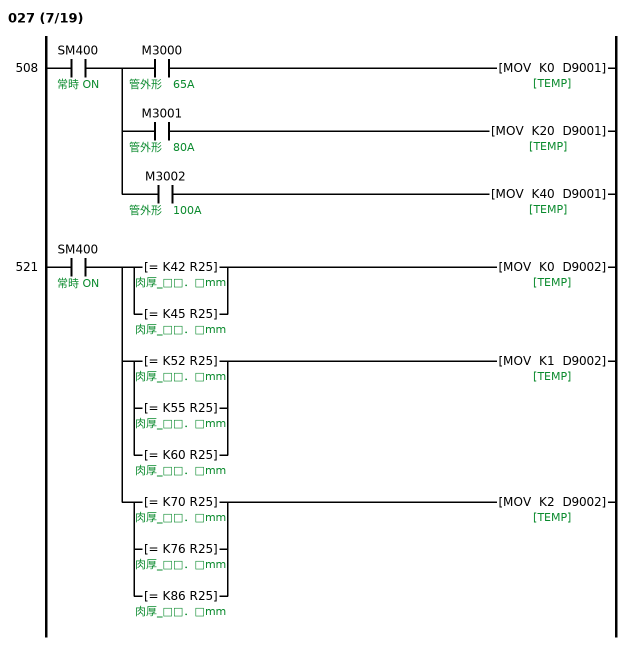
508   LD      SM400  ; 常時 ON
      MPS
      AND     M3000  ; 管外形　65A
      MOV     K0 D9001  ; [TEMP]
      MRD
      AND     M3001  ; 管外形　80A
      MOV     K20 D9001
      MPP
      AND     M3002  ; 管外形　100A
      MOV     K40 D9001
521   LD      SM400  ; 常時 ON
      MPS
      LD=     K42 R25  ; 肉厚_□□．□mm
      OR=     K45 R25  ; 肉厚_□□．□mm
      ANB
      MOV     K0 D9002
      MRD
      LD=     K52 R25  ; 肉厚_□□．□mm
      OR=     K55 R25  ; 肉厚_□□．□mm
      OR=     K60 R25  ; 肉厚_□□．□mm
      ANB
      MOV     K1 D9002
      MPP
      LD=     K70 R25  ; 肉厚_□□．□mm
      OR=     K76 R25  ; 肉厚_□□．□mm
      OR=     K86 R25  ; 肉厚_□□．□mm
      ANB
      MOV     K2 D9002
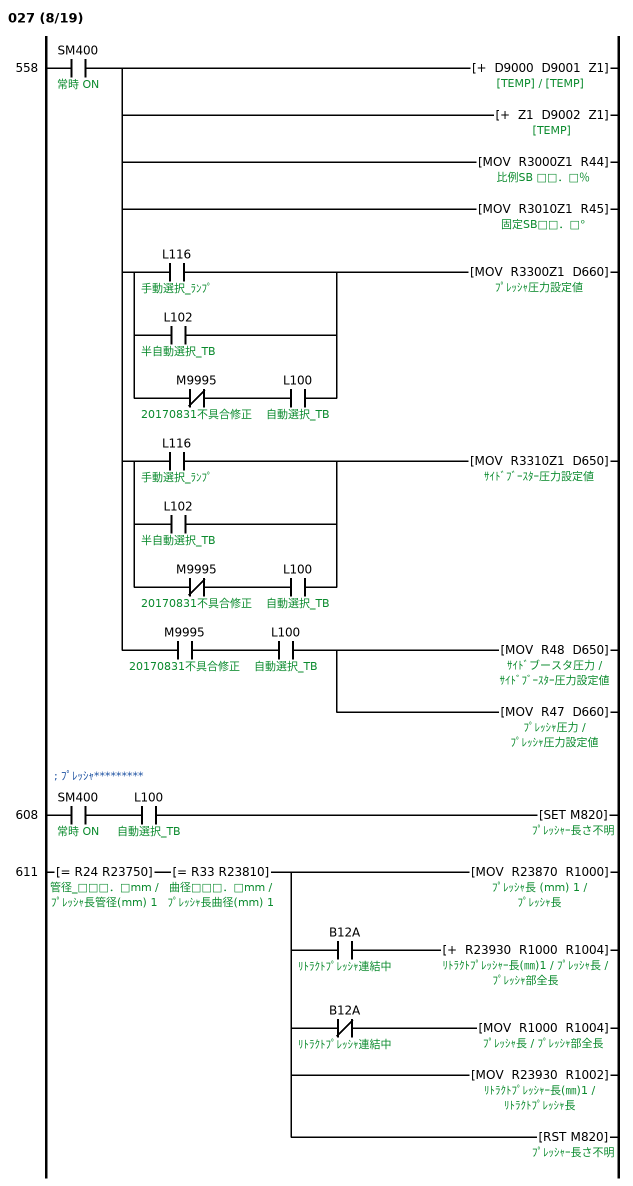
558   LD      SM400  ; 常時 ON
      +       D9000 D9001 Z1
      +       Z1 D9002 Z1
      MOV     R3000Z1 R44  ; 比例SB □□．□％
      MOV     R3010Z1 R45  ; 固定SB□□．□°
      MPS
      LD      L116  ; 手動選択_ﾗﾝﾌﾟ
      OR      L102  ; 半自動選択_TB
      LDI     M9995  ; 20170831不具合修正
      AND     L100  ; 自動選択_TB
      ORB
      ANB
      MOV     R3300Z1 D660  ; ﾌﾟﾚｯｼｬ圧力設定値
      MRD
      LD      L116  ; 手動選択_ﾗﾝﾌﾟ
      OR      L102  ; 半自動選択_TB
      LDI     M9995  ; 20170831不具合修正
      AND     L100  ; 自動選択_TB
      ORB
      ANB
      MOV     R3310Z1 D650  ; ｻｲﾄﾞﾌﾞｰｽﾀｰ圧力設定値
      MPP
      AND     M9995  ; 20170831不具合修正
      AND     L100  ; 自動選択_TB
      MOV     R48 D650  ; ｻｲﾄﾞブースタ圧力
      MOV     R47 D660  ; ﾌﾟﾚｯｼｬ圧力
; ﾌﾟﾚｯｼｬ*********
608   LD      SM400  ; 常時 ON
      AND     L100  ; 自動選択_TB
      SET     M820  ; ﾌﾟﾚｯｼｬｰ長さ不明
611   LD=     R24 R23750  ; 管径_□□□．□mm / ﾌﾟﾚｯｼｬ長管径(mm) 1
      AND=    R33 R23810  ; 曲径□□□．□mm / ﾌﾟﾚｯｼｬ長曲径(mm) 1
      MOV     R23870 R1000  ; ﾌﾟﾚｯｼｬ長 (mm) 1 / ﾌﾟﾚｯｼｬ長
      MPS
      AND     B12A  ; ﾘﾄﾗｸﾄﾌﾟﾚｯｼｬ連結中
      +       R23930 R1000 R1004  ; ﾘﾄﾗｸﾄﾌﾟﾚｯｼｬｰ長(㎜)1 / ﾌﾟﾚｯｼｬ部全長
      MRD
      ANI     B12A  ; ﾘﾄﾗｸﾄﾌﾟﾚｯｼｬ連結中
      MOV     R1000 R1004
      MPP
      MOV     R23930 R1002  ; ﾘﾄﾗｸﾄﾌﾟﾚｯｼｬ長
      RST     M820  ; ﾌﾟﾚｯｼｬｰ長さ不明
